Fanuc TP program (LS listing): HOME_POSITION.LS

/PROG  HOME_POSITION
/ATTR
OWNER		= MNEDITOR;
COMMENT		= "";
PROG_SIZE	= 516;
CREATE		= DATE 25-07-13  TIME 21:52:34;
MODIFIED	= DATE 25-07-13  TIME 21:56:16;
FILE_NAME	= ;
VERSION		= 0;
LINE_COUNT	= 4;
MEMORY_SIZE	= 872;
PROTECT		= READ_WRITE;
TCD:  STACK_SIZE	= 0,
      TASK_PRIORITY	= 50,
      TIME_SLICE	= 0,
      BUSY_LAMP_OFF	= 0,
      ABORT_REQUEST	= 0,
      PAUSE_REQUEST	= 0;
DEFAULT_GROUP	= 1,*,*,*,*;
CONTROL_CODE	= 00000000 00000000;
LOCAL_REGISTERS	= 0,0,0;
/APPL

LINE_TRACK;
  LINE_TRACK_SCHEDULE_NUMBER      : 0;
  LINE_TRACK_BOUNDARY_NUMBER      : 0;
  CONTINUE_TRACK_AT_PROG_END      : TRUE;

/MN
   1:  UFRAME_NUM=1 ;
   2:  UTOOL_NUM=1 ;
   3:   ;
   4:J P[1] 100% FINE    ;
/POS
P[1]{
   GP1:
	UF : 1, UT : 1,		CONFIG : 'N U T, 0, 0, 0',
	X =  -588.676  mm,	Y =      .196  mm,	Z =   306.969  mm,
	W =   180.000 deg,	P =     -.000 deg,	R =     -.000 deg
};
/END
